# EPICS StreamDevice protocol: vacApp/Db/QPC-serial.proto
# This protocol file ignores the checksum going to and from
# the device. It has been tested on QPC and MPCq but will likely
# also work for MPC as well.
OutTerminator = CR;
InTerminator = CR;
ReadTimeout = 2000;
ReplyTimeout = 2000;

# Command 0A Read Current
getCurrent {
	out "~ 05 0A \$1 00 ";
	in "%*9c%E %*7c";

	@mismatch { in "%(\$2\$3:Supply\$1StatusM.VAL)36c";}
}

# Command 0B Read Pressure
getPressure {
	out "~ 05 0B \$1 00 ";
	in "%*9c%E %*7c";

	@mismatch { in "%(\$2\$3:Supply\$1StatusM.VAL)36c";}
}

# Command 0C Read Voltage
getVoltage {
	out "~ 05 0C \$1 00";
	in "%*9c%d %*5c";

	@mismatch { in "%(\$2\$3:Supply\$1StatusM.VAL)36c";}
}

# Command 0D Get Supply Status
# New command has the format cmd 0D supply,option
# If you send cmd 0D \$1,00 (Currently 00 is the only option)
# The return format will be XX where XX is one of:
# 00 - pump standby
# 01 - pump starting
# 02 - pump running
# 03 - pump cooldown
# 04 - pump error
# Otherwise this protocol sends back a string as is done here
getStatus {
	out "~ 05 0D \$1 00";
	in "%*9c%s %*5c";
}

# Command 61 Is High Voltage On - Indicates if the high voltage is on for
# the specified pump
# This is likely a legacy command as it does not exist in the revision G
# manual. I think that it is replaced by the 0D command above.
isEnabled {
	out "~ 05 61 \$1 00";
	in "%*9c%s %*2c";

	@mismatch { in "%(\$2\$3:Supply\$1StatusM.VAL)36c";}
}

# Command 37 Start Pump - Enables high voltage of specified supply
enable {
	out "~ 05 37 \$1 00";
}

# Command 38 Stop Pump - Disables high voltage of specified supply
disable {
	out "~ 05 38 \$1 00";
}

# Command 01 Get Model - Returns the pump controller model (QPC,MPC,etc)
getModel {
	out "~ 05 01 00";
	in "%*17c%s %*2c";
}

# Command 02 Version - Returns the firmware version of the pump controller
getFirmware {
	out "~ 05 02 00";
	in "%*27c%s %*2c";
}

# This function is used to initialize setPressUnit function below
getPressureUnit {
	out "~ 05 0B \$1 00";
	in "%*9c%*f%*1c%s %*2X";
}

# Uses the command 0B above but returns only the pressure units selected
# Command 0E Set Pressure Units - Allows remote control over pressure units
setPressUnit {
	out "~ 05 0E %s\$1 00";
	in "%*11c";

#	@init { getPressureUnit; }
}

# Command 11 Get pump Size - Reads pump size in liters/second
getPumpSize {
	out "~ 05 11 \$1 00";
	in "%*9c%d L/S %*2X";
}

# Command 12 Set pump Size - Sets pump size in liters/second
setPumpSize {
	out "~ 05 12 \$1,%s 00";
	in "%*9c";
}

# For the set points here we just get the set point on/off pressure and output
# relay/digital out status
# NOTE:
# We will use the new 3B command which has replaced the 3C and 3D commands
# get the on pressure set point
# Response from 3B command
# 05 OK 00 1,1,1,3.0E-08,3.6E-08,1 5B
# Response format:
# ADDR STATUS ERR DATA CHECKSUM
# DATA is: (See QPC manual version L pg 47)
# Spt#,Func,Supply#,On Pressure, Off Pressure
# Func can be one of: 0-Off, 1-On, 2-HV Error, 3-HV On/Off Indicator
getPressSpt {
	out "~ 05 3B \$1 00";
	in "%*14c,%(\$2\$3:Spt\$1OnPressM.VAL)E,%(\$2\$3:Spt\$1OffPressM.RVAL)E,%(\$2\$3:Spt\$1StatusM.RVAL)d%*3c";

	@mismatch { in "%(\$2\$3:Supply\$1StatusM.VAL)36c";}
}

# The mismatch is because I got lazy with the database and did not filter
# bad on pressures being sent to the device mostly because the device
# firmware will automatically set the off pressure 20% > than the on pressure.
setOffPress {
	out "~ 05 3B \$2,1,\$1,%E,%(\$3\$4:Spt\$2OffPressM.VAL)E 00";
	in "%*17c%(\$3\$4:SptMessage.VAL)39c";

	@mismatch { in "ER 08 *ERROR: %(\$3\$4:SptMessage.VAL)36c";}
}
setOnPress {
	out "~ 05 3B \$2,1,\$1,%(\$3\$4:Spt\$2OnPressM.VAL)E,%E 00";
	in "%*11c";
}

# Pump (supply) name is 15 characters max.
getPumpName {
	out "~ 05 ED \$1 00";
	in "%*9c%15s %*4c";
}

# Get Auto Restart Status for Supply
getAutoRestart {
	out "~ 05 34 \$1 00";
	in "05 OK 00 %s %*2c";
}

# Set Auto Restart Status for Supply
setAutoRestart {
	out "~ 05 33 \$1,%s 00";
}
